FUNCTION_BLOCK FINAL AdsLogSink IMPLEMENTS ITcoLogSink
VAR_INPUT
END_VAR
VAR_OUTPUT
END_VAR
VAR
END_VAR

METHOD Emit : BOOL
VAR_INPUT
	LogEvent	: REFERENCE TO LogEvent;
END_VAR
IF NOT __ISVALIDREF(LogEvent) THEN
	RETURN;
END_IF

// ADSLOGSTR(0, LogEvent.Text, '');
END_METHOD

END_FUNCTION_BLOCK

(* stored: Version 1.1.0.1, ProductVersion 3.1.4024.9
   POU AdsLogSink: Id {d9931d1f-35a0-0c3e-16a4-d9f0f4bf0e4a}, SpecialFunc None
   Method Emit: Id {abc98689-d825-0286-2b15-2a7963025d80} *)
